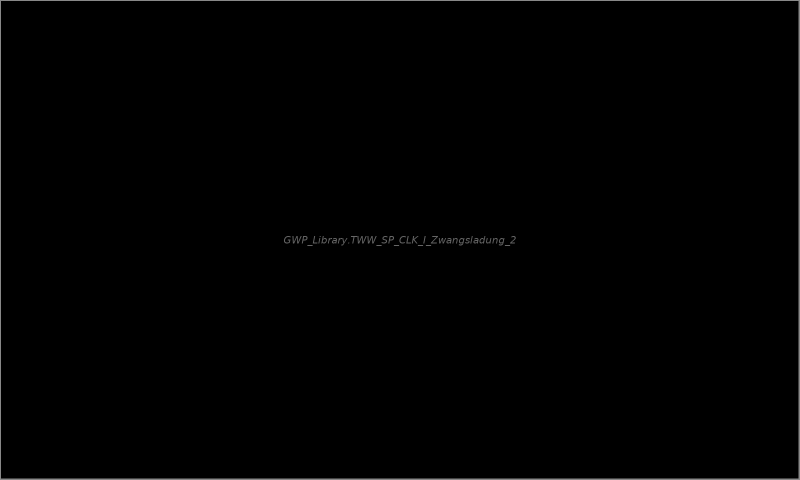
VISUALIZATION TWW_SP_CLK_I_Zwangsladung_2  // 800x480
    Frame (0,0 800x480)
        shows GWP_Library.TWW_SP_CLK_I_Zwangsladung_2(FB_CLK_I := Main.TWW_SP_0.CLK_I_1, FB_Init_1 := Main.Init_0)
END_VISUALIZATION

(* stored: Version 1.1.0.1, ProductVersion 3.1.4022.6
   Visu TWW_SP_CLK_I_Zwangsladung_2: Id {b477f942-c58d-4c58-bd54-8ede2b681d16} *)
